# EPICS substitutions: ecmcApp/Db/SlitX-xl-extra.substitutions
file "ecmc-extra.template"
{
pattern
{P,      M,    R,   PORT, ADDR, PREC, HOMEPROC}
{IOC2:,  xl, xl-,   MCU1,    3, 3,    3}
}
